# EPICS substitutions: GalilTestApp/Db/galil_motor.substitutions
# $File: //ASP/Dev/SBS/4_Controls/4_3_Network_Infrastructure/4_3_1_Comms_Common_Services/sw/device_drivers/Galil/1-5/galilTestApp/Db/galil_motor_withwrappers.substitutions $
# $Revision: #3 $
# $DateTime: 2012/03/22 09:46:31 $
# $Author: cliftm $
#
# Description
# Substitution file for motor_withwrappers.template
#
# MOVNFLNK FLNK when moving status is updated
# LIMITFLNK FLNK when limits are updated
# READBACK used to set read back to user or dial coordinates
#
# This library is free software; you can redistribute it and/or
# modify it under the terms of the GNU Lesser General Public
# Licence as published by the Free Software Foundation; either
# version 2.1 of the Licence, or (at your option) any later version.
#
# This library is distributed in the hope that it will be useful,
# but WITHOUT ANY WARRANTY; without even the implied warranty of
# MERCHANTABILITY or FITNESS FOR A PARTICULAR PURPOSE.  See the GNU
# Lesser General Public Licence for more details.
#
# You should have received a copy of the GNU Lesser General Public
# Licence along with this library; if not, write to the Free Software
# Foundation, Inc., 51 Franklin St, Fifth Floor, Boston, MA 02110-1301 USA.
#
# Contact details:
# mark.clift@synchrotron.org.au
# 800 Blackburn Road, Clayton, Victoria 3168, Australia.
#

file "$(GALIL)/GalilSup/Db/galil_motor.template"
{
pattern
{   P,       M,   PORT,    ADDR, EGU, DESC, VELO,  VMAX,  ACCL,  BDST,  BVEL,  BACC,  MRES,  SREV, ERES,     PREC, DHLM,    DLLM,     OFF,     UEIP, RTRY, PCOF, ICOF, DCOF}

# Real motors
   {"\$(P)", "MTR$(CCP)01", "Galil", 0,    mm,  "",   20,    20,    1,     0,     0,     5,     .0025, 1000, 0.000625, 5,    42273.3, -42273.3, 0,       0,    0   , 0,    0,    0}
   {"\$(P)", "MTR$(CCP)02", "Galil", 1,    mm,  "",   .2,    .2,    1,     0,     0,     5,     .0025, 1000, 0.000625, 5,    42273.3, -42273.3, 0,       0,    0   , 0,    0,    0}
   {"\$(P)", "MTR$(CCP)03", "Galil", 2,    mm,  "",   .2,    .2,    1,     0,     0,     5,     .0025, 400,  0.001,    5,    42273.3, -42273.3, 0,       0,    0   , 0,    0,    0}
   {"\$(P)", "MTR$(CCP)04", "Galil", 3,    mm,  "",   .2,    .2,    1,     0,     0,     5,     .0025, 400,  0.001,    5,    42273.3, -42273.3, 0,       0,    0   , 0,    0,    0}
   {"\$(P)", "MTR$(CCP)05", "Galil", 4,    mm,  "",   .2,    .2,    1,     0,     0,     5,     .0025, 400,  0.001,    5,    42273.3, -42273.3, 0,       0,    0   , 0,    0,    0}
   {"\$(P)", "MTR$(CCP)06", "Galil", 5,    mm,  "",   .2,    .2,    1,     0,     0,     5,     .0025, 400,  0.001,    5,    42273.3, -42273.3, 0,       0,    0   , 0,    0,    0}
   {"\$(P)", "MTR$(CCP)07", "Galil", 6,    mm,  "",   .2,    .2,    1,     0,     0,     5,     .0025, 400,  0.001,    5,    42273.3, -42273.3, 0,       0,    0   , 0,    0,    0}
   {"\$(P)", "MTR$(CCP)08", "Galil", 7,    mm,  "",   .2,    .2,    1,     0,     0,     5,     .0025, 400,  0.001,    5,    42273.3, -42273.3, 0,       0,    0   , 0,    0,    0}

# Virtual motors
   {"\$(P)", "MTR$(CCP)09", "Galil", 8,    mm,  "",   20,    20,    1,     0,     0,     5,     .0025, 1000, 0.000625, 5,    42273.3, -42273.3, 0,       0,    0   , 0,    0,    0}
   {"\$(P)", "MTR$(CCP)10", "Galil", 9,    mm,  "",   20,    20,    1,     0,     0,     5,     .0025, 1000, 0.000625, 5,    42273.3, -42273.3, 0,       0,    0   , 0,    0,    0}

}

# end
